{attribute 'GeneratedUsingTerminal: EL7211-0010-0032'}
{attribute addProperty BoxType "EL7211-0010-0032"}
{attribute addProperty Id "Target_positionAT %Q*UDINT4"}
{attribute addProperty CRC "86249236"}
{attribute addProperty Size "4"}
TYPE DRV_Target_position_05240F14 EXTENDS TcoIo.OutputBase_10CEE7DE :
STRUCT
	{attribute addProperty Name "Target_position"}
	Target_position AT %Q* : UDINT;
END_STRUCT
END_TYPE

(* stored: Version 1.2.0.0, ProductVersion 3.1.4024.11
   DUT DRV_Target_position_05240F14: Id {f7275695-790e-08d0-1771-587d374aba8f} *)
